"CYC_INT2"	OB 32	OB 32	// CYCLIC INTERRUPT 2
"CYC_INT4"	OB 34	OB 34	// CYCLIC INTERRUPT 4
"I/O_FLT1"	OB 82	OB 82	// I/O POINT FAULT 1
"I/O_FLT2"	OB 83	OB 83	// I/O POINT FAULT 2
"OBNL_FLT"	OB 85	OB 85	// OB NOT LOADED FAULT
"RACK_FLT"	OB 86	OB 86	// LOSS OF RACK FAULT
"COMM_FLT"	OB 87	OB 87	// Communication Fault
"COMPLETE RESTART"	OB 100	OB 100	// COMPLETE RESTART
"MOD_ERR"	OB 122	OB 122	// Module Access Error
"VADI"	Q 0.0	BOOL	// (MOP-IM.M06-07): LAMPARA ANULACION DEFECTO
"VMCY"	Q 0.1	BOOL	// (MOP-IM.M06-07): LAMPARA MARCHA CICLO
"VAOP"	Q 0.3	BOOL	// (MOP-IM.M06-07): BALIZA LLAMADA OPERARIO
"Alas"	Q 2.0	BOOL	// ALARMA SONORA
"AlaL"	Q 2.1	BOOL	// ALARMA LUMINOSA
"Z1VMCY"	Q 100.0	BOOL	// (Z1ZB.M04): CYCLE START LAMP
"Z1VDINJ"	Q 100.1	BOOL	// (Z1ZB.M04): LAMPADA INYECCION SIPTOL
"Z1RCM"	Q 100.7	BOOL	// (Z1ZB.M04): RELE DE MASA
"Z1RFRO1"	Q 108.0	BOOL	// (Z1ZB.M07): COMUN DE SECURIDAD 1 (Z1AU)
"Z1RFRO2"	Q 108.1	BOOL	// (Z1ZB.M07): COMUN DE SECURIDAD 2 (Z1ES)
"Z1EV7B"	Q 108.3	BOOL	// (Z1ZB.M07): EV 7 BARS
"Z1RSC1"	Q 115.0	BOOL	// (Z1ZB.M09): RELE COMUN DE SEGURIDAD SC1
"Z1RES"	Q 115.1	BOOL	// (Z1ZB.M09): RELE COMUN DE SEGURIDAD ES
"Z1RFZ"	Q 115.2	BOOL	// (Z1ZB.M09): RELE COMUN DE SEGURIDAD FZ
"Z1RSC4"	Q 115.3	BOOL	// (Z1ZB.M09): RELE COMUN DE SEGURIDAD SC4
"A01VAT"	Q 201.0	BOOL	// LAMPADA AUTORIZACION DE TRABAJO OPERARIO (VERDE)
"A01VIT"	Q 201.1	BOOL	// VERINE INTERDICTION TRAVAIL (ROUGE)
"A01VDF"	Q 201.2	BOOL	// LAMPADA DEFECTO (NARANJA)
"A01VROC"	Q 201.3	BOOL	// LAMPADA ORIGEN DE CYCLO
"A01RFRO1"	Q 220.0	BOOL	// RELE DE SECURIDAD OPERARIO
"A01RFRO2"	Q 220.1	BOOL	// Commun de sécurité 4 (F-RO2 )
"A01RFRO3"	Q 220.2	BOOL	// Commun de sécurité 5 (F-RO3 )
"A0CCVB"	Q 225.4	BOOL	// ACCIONAM CILINDRO CAMBIO DE VIA B52
"A0CCVL"	Q 225.5	BOOL	// ACCIONAM CILINDRO CAMBIO DE VIA L52
"B01VAT"	Q 231.0	BOOL	// LAMPADA AUTORIZACION DE TRABAJO OPERARIO (VERDE)
"B01VIT"	Q 231.1	BOOL	// LAMPADA INTERDICTION DE TRABAJO OPERARIO (ROJO)
"B01VDF"	Q 231.2	BOOL	// LAMPADA DEFECTO (NARANJA)
"B01VROC"	Q 231.3	BOOL	// LAMPADA ORIGEN DE CYCLO
"B01RFRO1"	Q 250.0	BOOL	// RELE DE SECURIDAD OPERARIO
"B01RFRO2"	Q 250.1	BOOL	// B01 SAFETY COMMUN
"B01RFRO3"	Q 250.2	BOOL	// B01 SAFETY COMMUN
"C01VAT"	Q 261.0	BOOL	// LAMPADA AUTORIZACION DE TRABAJO OPERARIO (VERDE)
"C01VIT"	Q 261.1	BOOL	// LAMPADA INTERDICTION DE TRABAJO OPERARIO (ROJO)
"C01VDF"	Q 261.2	BOOL	// LAMPADA DEFECTO (NARANJA)
"C01VROC"	Q 261.3	BOOL	// LAMPADA ORIGEN DE CYCLO
"C01RFRO1"	Q 280.0	BOOL	// RELE DE SECURIDAD OPERARIO
"C01RFRO2"	Q 280.1	BOOL	// C01 SAFETY COMMON
"C01RFRO3"	Q 280.2	BOOL	// C01 SAFETY COMMON
"B02VAT"	Q 291.0	BOOL	// LAMPADA AUTORIZACION DE TRABAJO OPERARIO (VERDE)
"B02VIT"	Q 291.1	BOOL	// LAMPADA INTERDICTION DE TRABAJO OPERARIO (ROJO)
"B02VDF"	Q 291.2	BOOL	// LAMPADA DEFECTO (NARANJA)
"B02VROC"	Q 291.3	BOOL	// LAMPADA ORIGEN DE CYCLO
"B02RFRO1"	Q 310.0	BOOL	// RELE DE SECURIDAD OPERARIO
"B02RFRO2"	Q 310.1	BOOL	// Commun de sécurité 4 (F-RO2 )
"B02RFRO3"	Q 310.2	BOOL	// Commun de sécurité 5 (F-RO3 )
"C02VAT"	Q 321.0	BOOL	//  VERINE CONTROLE  AUTORISATION (VERT)
"C02VIT"	Q 321.1	BOOL	// LAMPADA INTERDICTION DE TRABAJO OPERARIO (ROJO)
"C02VDF"	Q 321.2	BOOL	// LAMPADA DEFECTO (NARANJA)
"C02VROC"	Q 321.3	BOOL	// LAMPADA ORIGEN DE CYCLO
"C02RFRO1"	Q 340.0	BOOL	// RELE DE SECURIDAD OPERARIO
"C02RFRO2"	Q 340.1	BOOL	// C02 SAFETY COMMON
"C02RFRO3"	Q 340.2	BOOL	// C02 SAFETY COMMON
"A01EEPLA"	Q 420.0	BOOL	// A01 EV. RETROCESO PILOTO A
"A01EDPLA"	Q 420.1	BOOL	// A01 EV. AVANCE PILOTO A
"A01EDPLB"	Q 420.2	BOOL	// A01 EV. RETROCESO PILOTO B
"A01EEPLB"	Q 420.3	BOOL	// A01 EV. AVANCE PILOTO B
"A01EDPLC"	Q 420.4	BOOL	// A01 EV. RETROCESO PILOTO C
"A01EEPLC"	Q 420.5	BOOL	// A01 EV. AVANCE PILOTO C
"A01EDPLD"	Q 420.6	BOOL	// A01 EV. RETROCESO PILOTO D
"A01EEPLD"	Q 420.7	BOOL	// A01 EV. AVANCE PILOTO D
"A01NEEPLA"	Q 421.0	BOOL	// A01 EV. RETROCESO PILOTO A
"A01NEDPLA"	Q 421.1	BOOL	// A01 EV. AVANCE PILOTO A
"A01NEDPLB"	Q 421.2	BOOL	// A01 EV. RETROCESO PILOTO B
"A01NEEPLB"	Q 421.3	BOOL	// A01 EV. AVANCE PILOTO B
"A01NEDPLC"	Q 421.4	BOOL	// A01 EV. RETROCESO PILOTO C
"A01NEEPLC"	Q 421.5	BOOL	// A01 EV. AVANCE PILOTO C
"A01NEDPLD"	Q 421.6	BOOL	// A01 EV. RETROCESO PILOTO D
"A01NEEPLD"	Q 421.7	BOOL	// A01 EV. AVANCE PILOTO D
"A01EESRE"	Q 422.0	BOOL	// A01 EV. AVANCE APRIETE E
"A01EDSRE"	Q 422.1	BOOL	// A01 EV. RETROCESO APRIETE E
"A01EESRF"	Q 422.2	BOOL	// A01 EV. AVANCE APRIETE F
"A01EDSRF"	Q 422.3	BOOL	// A01 EV. RETROCESO APRIETE F
"A01EESRG"	Q 422.4	BOOL	// A01 EV. AVANCE APRIETE G
"A01EDSRG"	Q 422.5	BOOL	// A01 EV. RETROCESO APRIETE G
"A01EESRM"	Q 422.6	BOOL	// A01 EV. AVANCE APRIETE M
"A01EDSRM"	Q 422.7	BOOL	// A01 EV. RETROCESO APRIETE M
"A01EDSRH"	Q 425.0	BOOL	// A01 EV. RETROCESO APRIETE H
"A01EESRH"	Q 425.1	BOOL	// A01 EV. AVANCE APRIETE H
"A01EEEJL"	Q 425.2	BOOL	// A01 EV. AVANCE EYECTOR L
"A01EDEJL"	Q 425.3	BOOL	// A01 EV. RETROCESO EYECTOR L
"A01NEDSRH"	Q 441.0	BOOL	// A01 EV. RETROCESO APRIETE H
"A01NEESRH"	Q 441.1	BOOL	// A01 EV. AVANCE APRIETE H
"A01EESRJ"	Q 441.2	BOOL	// A01 EV. AVANCE APRIETE J
"A01EDSRJ"	Q 441.3	BOOL	// A01 EV. RETROCESO APRIETE J
"A01EESRK"	Q 441.4	BOOL	// A01 EV. AVANCE APRIETE K
"A01EDSRK"	Q 441.5	BOOL	// A01 EV. RETROCESO APRIETE K
"A01NEEEJL"	Q 441.6	BOOL	// A01 EV. AVANCE EYECTOR L
"A01NEDEJL"	Q 441.7	BOOL	// A01 EV. RETROCESO EYECTOR L
"B01EEPLA"	Q 480.0	BOOL	// B01 EV. AVANCE PILOTO A
"B01EDPLA"	Q 480.1	BOOL	// B01 EV. RETROCESO PILOTO A
"B01EEVTE"	Q 480.2	BOOL	// B01 EV. AVANCE VENTOSA E
"B01EDVTE"	Q 480.3	BOOL	// B01 EV. RETROCESO VENTOSA E
"B01EEEJK"	Q 480.6	BOOL	// B01 EV. AVANCE EYECTOR K
"B01EDEJK"	Q 480.7	BOOL	// B01 EV. RETROCESO EYECTOR K
"B01NEEPLA"	Q 481.0	BOOL	// B01 EV. AVANCE PILOTO A
"B01NEDPLA"	Q 481.1	BOOL	// B01 EV. RETROCESO PILOTO A
"B01EESRB"	Q 481.2	BOOL	// B01 EV. AVANCE APRIETE B
"B01EDSRB"	Q 481.3	BOOL	// B01 EV. RETROCESO APRIETE B
"B01EEPLC"	Q 481.4	BOOL	// B01 EV. AVANCE PILOTO C
"B01EDPLC"	Q 481.5	BOOL	// B01 EV. RETROCESO PILOTO C
"B01EEPLD"	Q 481.6	BOOL	// B01 EV. AVANCE PILOTO D
"B01EDPLD"	Q 481.7	BOOL	// B01 EV. RETROCESO PILOTO D
"1"	Q 482.0	BOOL
"2"	Q 482.1	BOOL
"B01EESRF"	Q 482.2	BOOL	// B01 EV. AVANCE APRIETE F
"B01EDSRF"	Q 482.3	BOOL	// B01 EV. RETROCESO APRIETE F
"B01EEAPC"	Q 482.6	BOOL	// B01 EV.AVANCE PILOTO CERRADURA
"B01EDRPC"	Q 482.7	BOOL	// B01 EV.RETROCESO PILOTO CERRADURA
"B01EESRG"	Q 501.0	BOOL	// B01 EV. AVANCE APRIETE G
"B01EDSRG"	Q 501.1	BOOL	// B01 EV. RETROCESO APRIETE G
"B01EESRH"	Q 501.2	BOOL	// B01 EV. AVANCE APRIETE H
"B01EDSRH"	Q 501.3	BOOL	// B01 EV. RETROCESO APRIETE H
"B01EESRJ"	Q 501.4	BOOL	// B01 EV. AVANCE APRIETE J
"B01EDSRJ"	Q 501.5	BOOL	// B01 EV. RETROCESO APRIETE J
"B01NEEEJK"	Q 501.6	BOOL	// B01 EV. AVANCE EYECTOR K
"B01NEDEJK"	Q 501.7	BOOL	// B01 EV. RETROCESO EYECTOR K
"C01EEPLA"	Q 540.0	BOOL	// C01 EV. AVANCE PILOTO A
"C01EDPLA"	Q 540.1	BOOL	// C01 EV. RETROCESO PILOTO A
"C01EEVTE"	Q 540.2	BOOL	// C01 EV. AVANCE VENTOSA E
"C01EDVTE"	Q 540.3	BOOL	// C01 EV. RETROCESO VENTOSA E
"C01EEEJJ"	Q 540.6	BOOL	// C01 EV. AVANCE EYECTOR J
"C01EDEJJ"	Q 540.7	BOOL	// C01 EV. RETROCESO EYECTOR J
"C01NEEPLA"	Q 541.0	BOOL	// C01 EV. AVANCE PILOTO A
"C01NEDPLA"	Q 541.1	BOOL	// C01 EV. RETROCESO PILOTO A
"C01EEABB"	Q 541.2	BOOL	// C01 EV. AVANCE APRIETE B
"C01EDABB"	Q 541.3	BOOL	// C01 EV. AVANCE APRIETE B
"C01EEPLC"	Q 541.4	BOOL	// C01 EV. AVANCE PILOTO C
"C01EDPLC"	Q 541.5	BOOL	// C01 EV. RETROCESO PILOTO C
"C01EEPLD"	Q 541.6	BOOL	// C01 EV. AVANCE PILOTO D
"C01EDPLD"	Q 541.7	BOOL	// C01 EV. RETROCESO PILOTO D
"C01EESRF"	Q 542.2	BOOL	// C01 EV. AVANCE APRIETE F
"C01EDSRF"	Q 542.3	BOOL	// C01 EV. RETROCESO APRIETE F
"C01EESRG"	Q 561.0	BOOL	// C01 EV. AVANCE APRIETE G
"C01EDSRG"	Q 561.1	BOOL	// C01 EV. RETROCESO APRIETE G
"C01EESRH"	Q 561.2	BOOL	// C01 EV. AVANCE APRIETE H
"C01EDSRH"	Q 561.3	BOOL	// C01 EV. RETROCESO APRIETE H
"C01NEEEJJ"	Q 561.4	BOOL	// C01 EV. AVANCE EYECTOR J
"C01NEDEJJ"	Q 561.5	BOOL	// C01 EV. RETROCESO EYECTOR J
"B02EDPLA"	Q 600.0	BOOL	// B02 EV. RETROCESO PILOTO A
"B02EEPLA"	Q 600.1	BOOL	// B02 EV. AVANCE PILOTO A
"B02EEVTE"	Q 600.2	BOOL	// accionar sopapa
"B02EDVTE"	Q 600.3	BOOL	// liberar sopapa
"B02EEEJL"	Q 600.6	BOOL	// B02 EV. AVANCE EYECTOR L
"B02EDEJL"	Q 600.7	BOOL	// B02 EV. RETROCESO EYECTOR L
"B02NEDPLA"	Q 601.0	BOOL	// B02 EV. RETROCESO PILOTO A
"B02NEEPLA"	Q 601.1	BOOL	// B02 EV. AVANCE PILOTO A
"B02EESRB"	Q 601.2	BOOL	// B02 EV. AVANCE APRIETE B
"B02EDSRB"	Q 601.3	BOOL	// B02 EV. RETROCESO APRIETE B
"B02EEPLC"	Q 601.4	BOOL	// B02 EV. AVANCE PILOTO C
"B02EDPLC"	Q 601.5	BOOL	// B02 EV. RETROCESO PILOTO C
"B02EEPLD"	Q 601.6	BOOL	// B02 EV. AVANCE PILOTO D
"B02EDPLD"	Q 601.7	BOOL	// B02 EV. RETROCESO PILOTO D
"B02EESRF"	Q 602.2	BOOL	// B02 EV. AVANCE APRIETE F
"B02EDSRF"	Q 602.3	BOOL	// B02 EV. RETROCESO APRIETE F
"B02EESRG"	Q 621.0	BOOL	// B02 EV. AVANCE APRIETE G
"B02EDSRG"	Q 621.1	BOOL	// B02 EV. RETROCESO APRIETE G
"B02EESRH"	Q 621.2	BOOL	// B02 EV. AVANCE APRIETE H
"B02EDSRH"	Q 621.3	BOOL	// B02 EV. RETROCESO APRIETE H
"B02EESRJ"	Q 621.4	BOOL	// B02 EV. AVANCE APRIETE J
"B02EDSRJ"	Q 621.5	BOOL	// B02 EV. RETROCESO APRIETE J
"B02EESRK"	Q 621.6	BOOL	// B02 EV. AVANCE APRIETE K
"B02EDSRK"	Q 621.7	BOOL	// B02 EV. RETROCESO APRIETE K
"B02NEEEJL"	Q 622.0	BOOL	// B02 EV. AVANCE EYECTOR L
"B02NEDEJL"	Q 622.1	BOOL	// B02 EV. RETROCESO EYECTOR L
"C02EDPLA"	Q 660.0	BOOL	// C02 EV. RETROCESO PILOTO A
"C02EEPLA"	Q 660.1	BOOL	// C02 EV. AVANCE PILOTO A
"C02EEVTD"	Q 660.2	BOOL	// C02 EV. AVANCE VENTOSA D
"C02EDVTD"	Q 660.3	BOOL	// C02 EV. RETROCESO VENTOSA D
"C02EEEJJ"	Q 660.6	BOOL	// C02 EV. AVANCE EYECTOR J
"C02EDEJJ"	Q 660.7	BOOL	// C02 EV. RETROCESO EYECTOR J
"C02NEDPLA"	Q 661.0	BOOL	// C02 EV. RETROCESO PILOTO A
"C02NEEPLA"	Q 661.1	BOOL	// C02 EV. AVANCE PILOTO A
"C02EEABB"	Q 661.2	BOOL	// C02 EV. AVANCE APRIETE B
"C02EDABB"	Q 661.3	BOOL	// C02 EV. RETROCESO APRIETE B
"C02EEPLC"	Q 661.4	BOOL	// C02 EV. AVANCE PILOTO C
"C02EDPLC"	Q 661.5	BOOL	// C02 EV. RETROCESO PILOTO C
"C02EESRE"	Q 662.0	BOOL	// C02 EV. AVANCE APRIETE E
"C02EDSRE"	Q 662.1	BOOL	// C02 EV. RETROCESO APRIETE E
"C02EESRF"	Q 662.2	BOOL	// C02 EV. AVANCE APRIETE F
"C02EDSRF"	Q 662.3	BOOL	// C02 EV. RETROCESO APRIETE F
"C02EESRG"	Q 680.0	BOOL	// C02 EV. AVANCE APRIETE G
"C02EDSRG"	Q 680.1	BOOL	// C02 EV. RETROCESO APRIETE G
"C02EESRH"	Q 680.2	BOOL	// C02 EV. AVANCE APRIETE H
"C02EDSRH"	Q 680.3	BOOL	// C02 EV. RETROCESO APRIETE H
"C02NEEEJJ"	Q 680.4	BOOL	// C02 EV. AVANCE EYECTOR J
"C02NEDEJJ"	Q 680.5	BOOL	// C02 EV. RETROCESO EYECTOR J
"TP"	SFB 3	SFB 3	// GENERATE A PULSE
"TON"	SFB 4	SFB 4	// GENERATE AN ON DELAY
"TOF"	SFB 5	SFB 5	// GENERATE AN OFF DELAY
"RDREC"	SFB 52	SFB 52	// READ A PROCESS DATA RECORD
"WRREC"	SFB 53	SFB 53	// WRITE A PROCESS DATA RECORD
"RALRM"	SFB 54	SFB 54	// Receive Alarm Data
"SET_CLK"	SFC 0	SFC 0	// SET SYSTEM CLOCK
"READ_CLK"	SFC 1	SFC 1	// READ SYSTEM CLOCK
"RD_SINFO"	SFC 6	SFC 6	// READ OB START INFORMATION
"D_ACT_DP"	SFC 12	SFC 12	// DEACTIVATING AND ACTIVATING DP SLAVES
"DPRD_DAT"	SFC 14	SFC 14	// READ CONSISTENT DATA OF A STANDARD DP SLAVE
"DPWR_DAT"	SFC 15	SFC 15	// WRITE CONSISTENT DATA TO A STANDARD DP SLAVE
"BLKMOV"	SFC 20	SFC 20	// COPY VARIABLES
"FILL"	SFC 21	SFC 21	// INITIALIZE A MEMORY AREA
"TEST_DB"	SFC 24	SFC 24	// TEST DATA BLOCK
"DIS_AIRT"	SFC 41	SFC 41	// DELAY THE HIGHER PRIORITY INTERRUPTS AND ASYNCHRONOUS ERRORS
"EN_AIRT"	SFC 42	SFC 42	// ENABLE HIGHER PRIORITY INTERRUPTS AND ASYNCHRONOUS ERRORS
"STP"	SFC 46	SFC 46	// CHANGE THE CPU TO STOP
"RDSYSST"	SFC 51	SFC 51	// READ A SYSTEM STATUS LIST OR PARTIAL LIST
"WR_REC"	SFC 58	SFC 58	// WRITE DATA RECORD
"RD_REC"	SFC 59	SFC 59	// READ A DATA RECORD
"TIME_TCK"	SFC 64	SFC 64	// READ THE SYSTEM TIME
"GEO_LOG"	SFC 70	SFC 70	// DETERMINE LOGICAL ADDRESS
"READ_DBL"	SFC 83	SFC 83	// READ DATA BLOCK OUT OF LOAD MEMORY
"WRIT_DBL"	SFC 84	SFC 84	// WRITE DATA BLOCK IN LOAD MEMORY
"DEL_SI"	SFC 106	SFC 106	// Deleting Dynamically Assigned System Instances
"ALARM_DQ"	SFC 107	SFC 107	// Creating Acknowledgeable Block-related Message
"ALARM_D"	SFC 108	SFC 108	// Creating Acknowledged Block-related Message
"C01TPE"	T 6	TIMER	// TEMP PIEC EJEC
"C02TPE"	T 7	TIMER	// TEMP PIEC EJEC
"pin"	T 8	TIMER	// pinchila
"T_C02PLC"	T 10	TIMER
"T_C01PLC"	T 11	TIMER
"TRMPPB02"	T 12	TIMER	// Tiempo para reset de MPP.MP.B02
"TRMPPB01"	T 13	TIMER	// Tiempo para reset de MPP.MP.B01
"TRMPPA01"	T 14	TIMER	// Tiempo para reset de MPP.MP.A01
"LIEN_SEC"	UDT 1507	UDT 1507
"IN_FONC"	UDT 1520	UDT 1520	// STANDARD HANDLING DRIVE'S IN FUNCTION CONTROL
"PILOTAGE"	UDT 1521	UDT 1521	// STANDARD HANDLING DRIVE'S CONTROL FUNCTION (FONC_VAR2)
"OUT_FONC"	UDT 1522	UDT 1522	// STANDARD HANDLING DRIVE'S OUT FUNCTION CONTROL (BF_FONC_VAR2)
"MOT_FONC_DPL"	UDT 1866	UDT 1866	// FUNCTION WORD FOR BF DP_LOCATOR USE / MOT FONCTION POUR LES BF DP_LOCATOR
"LIEN_TAB"	UDT 1936	UDT 1936
"LIEN_PUP"	UDT 1988	UDT 1988	// Gestion de modos y de pupitres de cde manu de la  ZONA (BF_ZONA_MODE_IHM)
"SL_IHM"	UDT 1999	UDT 1999
"LIEN_ILOT"	UDT 2004	UDT 2004	// INFO CONTROL LINKED TO THE FACILITY (BF_ILOT)
"MOT_FONC_MP"	UDT 2041	UDT 2041	// INFO CONTROL OF A MOVEMENT (BF_MOUVMP1)
"MOT_FONC"	UDT 2042	UDT 2042	// INFO DE UN MOUVIMIENTO(BF_MOUV2P1,BF_MVSE2P1, BF_RB_COD_PREH_API)
"FONC"	UDT 2047	UDT 2047
"VAT_1"	VAT 1	
"VAT_2"	VAT 2	
"SIPTOL_RECALAGE_C0R"	VAT 3	
"Palabra pieza  C01"	VAT 4	
"SIPTOL_ECH_A0L"	VAT 5	
"SIPTOL_ECH_B0L"	VAT 6	
"SIPTOL_ACQ_B0L"	VAT 7	
"SIPTOL_ACQ_A0L"	VAT 8	
"PUNTO_LANZAMIENTO"	VAT 9	
"Palabra pieza A01"	VAT 10	
"Palabra pieza  B01"	VAT 11	
"Palabra pieza  B02"	VAT 12	
"Palabra pieza  C02"	VAT 13	
"TEST_WAND"	VAT 14	
"SIPTOL_simple"	VAT 15	
"Presencias"	VAT 16	
END_SYMBOL_TABLE
